Omron CX-Programmer project NewProject (CX-Programmer 9.51)

# PLC TESTPLCOMRON: CJ1M CPU11

## Global symbols (name address type ; comment)
0.01 BOOL  ; Sent_Data_19
0.02 BOOL  ; Sent_Data_90
0.03 BOOL  ; Sent_Data_50
1.01 BOOL  ; Pump State
1.11 BOOL  ; Alarm
W0.00 BOOL  ; MOTOR ON
W0.01 BOOL  ; MOTOR OFF
W0.02 BOOL  ; ALARM ON
W0.03 BOOL  ; MOTOR ON
W0.04 BOOL  ; MOTOR OFF

## Program NewProgram1 (cyclic task 0)
Local symbols
DO UINT
LT101_Average D3303 UINT
L_LT_100cm W0.00 BOOL
Lim_Lvl_Hi #15E0 NUMBER
P_ON BOOL
Sent_Data_0 0.04 BOOL

### Section Section1

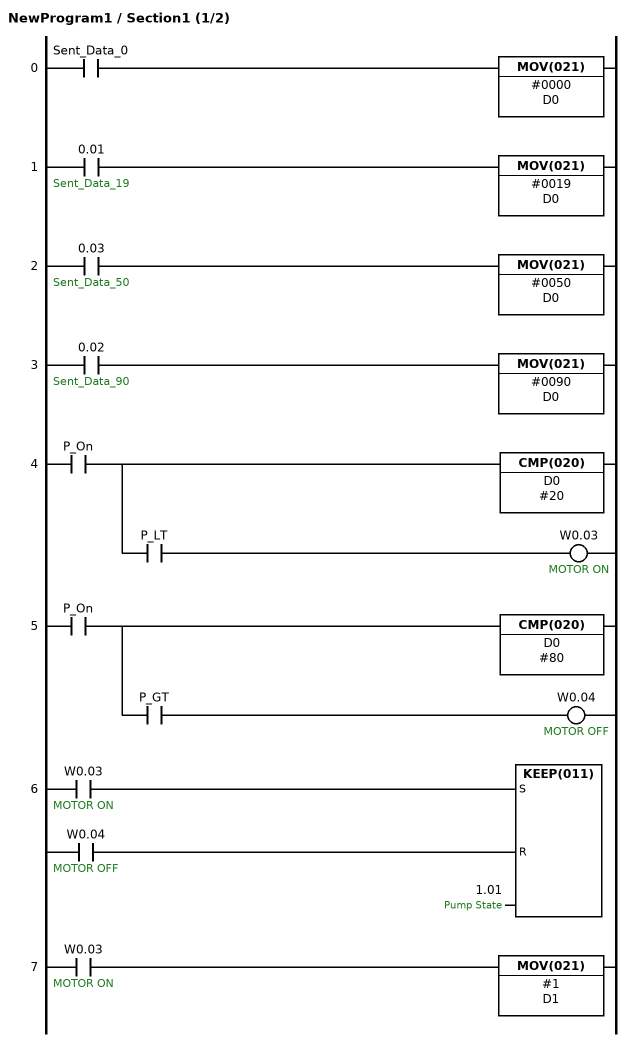
; rung 0
LD Sent_Data_0
MOV(021) #0000 D0
; rung 1
LD 0.01  ; Sent_Data_19
MOV(021) #0019 D0
; rung 2
LD 0.03  ; Sent_Data_50
MOV(021) #0050 D0
; rung 3
LD 0.02  ; Sent_Data_90
MOV(021) #0090 D0
; rung 4
LD P_On
CMP(020) D0 #20
AND P_LT
OUT W0.03  ; MOTOR ON
; rung 5
LD P_On
CMP(020) D0 #80
AND P_GT
OUT W0.04  ; MOTOR OFF
; rung 6
LD W0.03  ; MOTOR ON
LD W0.04  ; MOTOR OFF
KEEP(011) 1.01  ; Pump State
; rung 7
LD W0.03  ; MOTOR ON
MOV(021) #1 D1

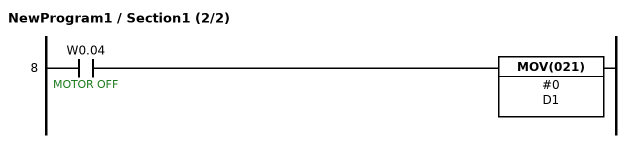
; rung 8
LD W0.04  ; MOTOR OFF
MOV(021) #0 D1

### Section END
; rung 0
END(001)